(* CoDeSys 2.3.9.44 project: Cap9_2.pro *)
(* Libraries: Standard.LIB 4.10.05 11:14:46 *)

(* Global variable list: Global_Variables *)
VAR_GLOBAL

(* Variables de entrada *)
    Numero: INT ;


(* Variables de Salida*)
      (* Siete segmentos de las centenas *)
      a0:BOOL;
	b0:BOOL;
	c0:BOOL;
	d0:BOOL;
	e0:BOOL;
	f0:BOOL;
	g0:BOOL;
      (* Siete segmentos de las decenas *)
      a1:BOOL;
	b1:BOOL;
	c1:BOOL;
	d1:BOOL;
	e1:BOOL;
	f1:BOOL;
	g1:BOOL;
   (* Siete segmentos de las unidades *)
      a2:BOOL;
	b2:BOOL;
	c2:BOOL;
	d2:BOOL;
	e2:BOOL;
	f2:BOOL;
	g2:BOOL;
      Novalido:BOOL;

END_VAR

(* POU PLC_PRG, ST *)
PROGRAM PLC_PRG
VAR
END_VAR

END_PROGRAM

(* Visualisation Display
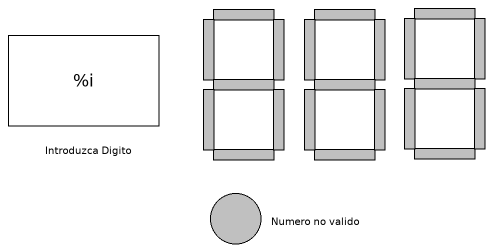
rectangle at (265,64)-(326,75): alarm colour if a0
rectangle at (325,74)-(336,135): alarm colour if b0
rectangle at (255,74)-(266,135): alarm colour if f0
rectangle at (265,134)-(326,145): alarm colour if g0
rectangle at (265,204)-(326,215): alarm colour if d0
rectangle at (325,144)-(336,205): alarm colour if c0
rectangle at (255,144)-(266,205): alarm colour if e0
rectangle at (60,90)-(211,181): text "%i"; shows Numero; editable
ellipse at (262,248)-(313,299): alarm colour if Novalido
rectangle at (60,190)-(221,221): text "Introduzca Digito"
rectangle at (287,261)-(448,292): text "Numero no valido"
rectangle at (366,64)-(427,75): alarm colour if a1
rectangle at (426,74)-(437,135): alarm colour if b1
rectangle at (356,74)-(367,135): alarm colour if f1
rectangle at (366,134)-(427,145): alarm colour if g1
rectangle at (366,204)-(427,215): alarm colour if d1
rectangle at (426,144)-(437,205): alarm colour if c1
rectangle at (356,144)-(367,205): alarm colour if e1
rectangle at (466,63)-(527,74): alarm colour if a2
rectangle at (526,73)-(537,134): alarm colour if b2
rectangle at (456,73)-(467,134): alarm colour if f2
rectangle at (466,133)-(527,144): alarm colour if g2
rectangle at (466,203)-(527,214): alarm colour if d2
rectangle at (526,143)-(537,204): alarm colour if c2
rectangle at (456,143)-(467,204): alarm colour if e2
*)
